// TIA Portal V20 program export: 1 tag tables, 0 data types, 2 data blocks, 4 code blocks (in call order from the OBs), 4 instance data blocks

VAR_GLOBAL   // PLC tag table "默认变量表"
   取芯V90_Actor_Interface_AddressIn AT %I82.0 : "PD_TEL3_IN";
   取芯V90_Actor_Interface_AddressOut AT %Q74.0 : "PD_TEL3_OUT";
   纠偏V90_Actor_Interface_AddressIn AT %I64.0 : "PD_TEL3_IN";
   纠偏V90_Actor_Interface_AddressOut AT %Q64.0 : "PD_TEL3_OUT";
   System_Byte AT %MB1 : Byte;
   FirstScan AT %M1.0 : Bool;
   DiagStatusUpdate AT %M1.1 : Bool;
   AlwaysTRUE AT %M1.2 : Bool;
   AlwaysFALSE AT %M1.3 : Bool;
   Clock_Byte AT %MB0 : Byte;
   Clock_10Hz AT %M0.0 : Bool;
   Clock_5Hz AT %M0.1 : Bool;
   "Clock_2.5Hz" AT %M0.2 : Bool;
   Clock_2Hz AT %M0.3 : Bool;
   "Clock_1.25Hz" AT %M0.4 : Bool;
   Clock_1Hz AT %M0.5 : Bool;
   "Clock_0.625Hz" AT %M0.6 : Bool;
   "Clock_0.5Hz" AT %M0.7 : Bool;
   纠偏V90控制字 AT %MW2 : Word;
   纠偏V90状态字 AT %MW4 : Word;
   纠_回原模式 AT %MW6 : Int;
   纠_绝对位置 AT %MD8 : Real;
   纠_相对位置 AT %MD12 : Real;
   纠_绝对速度 AT %MD16 : Real;
   纠_点动速度 AT %MD20 : Real;
   纠_当前位置 AT %M24.0 : LReal;
   纠_当前速度 AT %M32.0 : LReal;
   取芯V90控制字 AT %MW40 : Word;
   取芯V90状态字 AT %MW42 : Word;
   取_回原模式 AT %MW44 : Int;
   取_绝对位置 AT %MD46 : Real;
   取_绝对速度 AT %MD50 : Real;
   取_相对位置 AT %MD54 : Real;
   取_相对速度 AT %MD58 : Real;
   取_点动速度 AT %MD62 : Real;
   取_当前速度 AT %M66.0 : LReal;
   取_当前位置 AT %M74.0 : LReal;
END_VAR

DATA_BLOCK "G2_上传"   // DB2
{ S7_Optimized_Access := 'FALSE' }
   VAR
      位1 : Bool;
      位2 : Bool;
      位3 : Bool;
      位4 : Bool;
      位5 : Bool;
      位6 : Bool;
      位7 : Bool;
      位8 : Bool;
      位9 : Bool;
      位10 : Bool;
      位11 : Bool;
      位12 : Bool;
      位13 : Bool;
      位14 : Bool;
      位15 : Bool;
      位16 : Bool;
      位17 : Bool;
      位18 : Bool;
      位19 : Bool;
      位20 : Bool;
      位21 : Bool;
      位22 : Bool;
      位23 : Bool;
      位24 : Bool;
      位25 : Bool;
      位26 : Bool;
      位27 : Bool;
      位28 : Bool;
      位29 : Bool;
      位30 : Bool;
      整型1 : Int;
      整型2 : Int;
      整型3 : Int;
      整型4 : Int;
      整型5 : Int;
      整型6 : Int;
      整型7 : Int;
      整型8 : Int;
      整型9 : Int;
      整型10 : Int;
      浮点数1 : Real;
      浮点数2 : Real;
      浮点数3 : Real;
      浮点数4 : Real;
      浮点数5 : Real;
      浮点数6 : Real;
      浮点数7 : Real;
      浮点数8 : Real;
      浮点数9 : Real;
      浮点数10 : Real;
      浮点数11 : Real;
      浮点数12 : Real;
      浮点数13 : Real;
      浮点数14 : Real;
      浮点数15 : Real;
      浮点数16 : Real;
      浮点数17 : Real;
      浮点数18 : Real;
      浮点数19 : Real;
   END_VAR
BEGIN
END_DATA_BLOCK

DATA_BLOCK "G2_下载"   // DB1
{ S7_Optimized_Access := 'FALSE' }
   VAR
      位1 : Bool;
      位2 : Bool;
      位3 : Bool;
      位4 : Bool;
      位5 : Bool;
      位6 : Bool;
      位7 : Bool;
      位8 : Bool;
      位9 : Bool;
      位10 : Bool;
      位11 : Bool;
      位12 : Bool;
      位13 : Bool;
      位14 : Bool;
      位15 : Bool;
      位16 : Bool;
      位17 : Bool;
      位18 : Bool;
      位19 : Bool;
      位20 : Bool;
      位21 : Bool;
      位22 : Bool;
      位23 : Bool;
      位24 : Bool;
      位25 : Bool;
      位26 : Bool;
      位27 : Bool;
      位28 : Bool;
      位29 : Bool;
      位30 : Bool;
      整型1 : Int;
      整型2 : Int;
      整型3 : Int;
      整型4 : Int;
      整型5 : Int;
      整型6 : Int;
      整型7 : Int;
      整型8 : Int;
      整型9 : Int;
      整型10 : Int;
      浮点数1 : Real;
      浮点数2 : Real;
      浮点数3 : Real;
      浮点数4 : Real;
      浮点数5 : Real;
      浮点数6 : Real;
      浮点数7 : Real;
      浮点数8 : Real;
      浮点数9 : Real;
      浮点数10 : Real;
      浮点数11 : Real;
      浮点数12 : Real;
      浮点数13 : Real;
      浮点数14 : Real;
      浮点数15 : Real;
      浮点数16 : Real;
      浮点数17 : Real;
      浮点数18 : Real;
      浮点数19 : Real;
   END_VAR
BEGIN
END_DATA_BLOCK

ORGANIZATION_BLOCK "Main"   // OB1, LAD, ProgramCycle
TITLE = "Main Program Sweep (Cycle)"
{ S7_Optimized_Access := 'TRUE' }
// stored: SetENOAutomatically false
   VAR_INPUT
      Initial_Call : Bool;   // Initial call of this OB
      Remanence : Bool;   // =True, if remanent data are available
   END_VAR
BEGIN
END_ORGANIZATION_BLOCK

FUNCTION_BLOCK "定位轴基本控制"   // FB1, LAD
{ S7_Optimized_Access := 'TRUE' }
// stored: MemoryReserve 100, SetENOAutomatically false
   VAR_INPUT
      轴号 : TO_PositioningAxis;
      使能 : Bool;
      回原 : Bool;
      回原模式 : Int;
      绝对定位 : Bool;
      相对定位 : Bool;
      暂停 : Bool;
      复位 : Bool;
      绝对位置 : Real;
      绝对速度 : Real;
      相对位置 : Real;
      相对速度 : Real;
      点动正转 : Bool;
      点动反转 : Bool;
      点动速度 : Real;
   END_VAR
   VAR_OUTPUT
      轴已启用 : Bool;
      使能错误 : Bool;
      回原完成 : Bool;
      回原错误 : Bool;
      绝对定位完成 : Bool;
      绝对定位错误 : Bool;
      相对定位完成 : Bool;
      相对定位错误 : Bool;
      点动中 : Bool;
      点动错误 : Bool;
      当前位置 : LReal;
      当前速度 : LReal;
   END_VAR
   VAR
      MC_Power_Instance { S7_SetPoint := 'True'} : MC_POWER;
      MC_Home_Instance { S7_SetPoint := 'True'} : MC_HOME;
      MC_MoveAbsolute_Instance { S7_SetPoint := 'True'} : MC_MOVEABSOLUTE;
      MC_MoveRelative_Instance { S7_SetPoint := 'True'} : MC_MOVERELATIVE;
      MC_Reset_Instance { S7_SetPoint := 'True'} : MC_RESET;
      MC_Halt_Instance { S7_SetPoint := 'True'} : MC_HALT;
      MC_MoveJog_Instance { S7_SetPoint := 'True'} : MC_MOVEJOG;
   END_VAR
   VAR_TEMP
      复位完成 : Bool;
      复位错误 : Bool;
      暂停完成 : Bool;
      暂停错误 : Bool;
   END_VAR
   VAR_TEMP   // added for the SCL form of the ladder/FBD networks
      _w1 : Bool;
      _w2 : Bool;
      _w3 : Bool;
   END_VAR
BEGIN

REGION Network 1
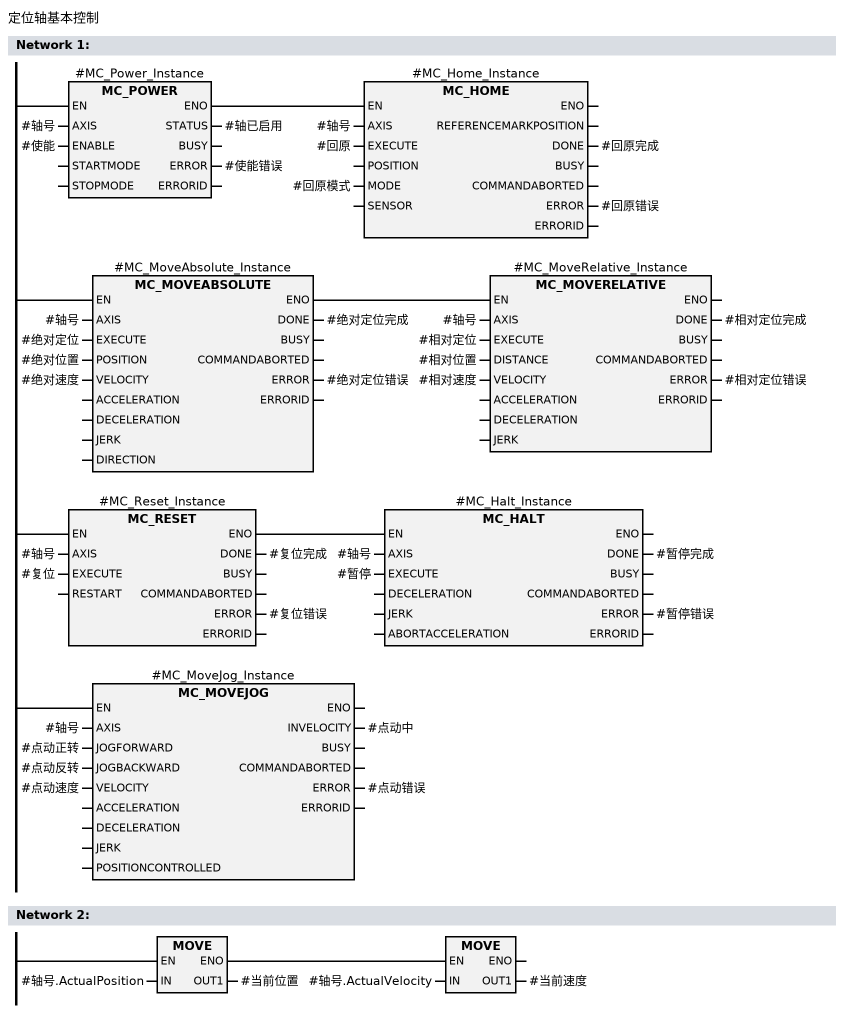
   RUNG wire#powerrail
      #MC_Power_Instance.MC_POWER(Axis := #轴号, Enable := #使能, StartMode :=, StopMode :=, Status => #轴已启用, Busy =>, Error => #使能错误, ErrorId =>)
      #MC_Home_Instance.MC_HOME(Axis := #轴号, Execute := #回原, Position :=, Mode := #回原模式, Sensor :=, ReferenceMarkPosition =>, Done => #回原完成, Busy =>, CommandAborted =>, Error => #回原错误, ErrorId =>)
   END_RUNG
   RUNG wire#powerrail
      #MC_MoveAbsolute_Instance.MC_MOVEABSOLUTE(Axis := #轴号, Execute := #绝对定位, Position := #绝对位置, Velocity := #绝对速度, Acceleration :=, Deceleration :=, Jerk :=, Direction :=, Done => #绝对定位完成, Busy =>, CommandAborted =>, Error => #绝对定位错误, ErrorId =>)
      #MC_MoveRelative_Instance.MC_MOVERELATIVE(Axis := #轴号, Execute := #相对定位, Distance := #相对位置, Velocity := #相对速度, Acceleration :=, Deceleration :=, Jerk :=, Done => #相对定位完成, Busy =>, CommandAborted =>, Error => #相对定位错误, ErrorId =>)
   END_RUNG
   RUNG wire#powerrail
      #MC_Reset_Instance.MC_RESET(Axis := #轴号, Execute := #复位, Restart :=, Done => #复位完成, Busy =>, CommandAborted =>, Error => #复位错误, ErrorId =>)
      #MC_Halt_Instance.MC_HALT(Axis := #轴号, Execute := #暂停, Deceleration :=, Jerk :=, AbortAcceleration :=, Done => #暂停完成, Busy =>, CommandAborted =>, Error => #暂停错误, ErrorId =>)
   END_RUNG
   RUNG wire#powerrail
      #MC_MoveJog_Instance.MC_MOVEJOG(Axis := #轴号, JogForward := #点动正转, JogBackward := #点动反转, Velocity := #点动速度, Acceleration :=, Deceleration :=, Jerk :=, PositionControlled :=, InVelocity => #点动中, Busy =>, CommandAborted =>, Error => #点动错误, ErrorId =>)
   END_RUNG
   // the same network as SCL:
   #MC_Power_Instance(Axis := #轴号, Enable := #使能, Status => #轴已启用, Error => #使能错误, ENO => #_w1);   // MC_POWER
   IF #_w1 THEN
       #MC_Home_Instance(Axis := #轴号, Execute := #回原, Mode := #回原模式, Done => #回原完成, Error => #回原错误);   // MC_HOME
   END_IF;
   #MC_MoveAbsolute_Instance(Axis := #轴号,   // MC_MOVEABSOLUTE
                           Execute := #绝对定位,
                           Position := #绝对位置,
                           Velocity := #绝对速度,
                           Done => #绝对定位完成,
                           Error => #绝对定位错误,
                           ENO => #_w2);
   IF #_w2 THEN
       #MC_MoveRelative_Instance(Axis := #轴号,   // MC_MOVERELATIVE
                               Execute := #相对定位,
                               Distance := #相对位置,
                               Velocity := #相对速度,
                               Done => #相对定位完成,
                               Error => #相对定位错误);
   END_IF;
   #MC_Reset_Instance(Axis := #轴号, Execute := #复位, Done => #复位完成, Error => #复位错误, ENO => #_w3);   // MC_RESET
   IF #_w3 THEN
       #MC_Halt_Instance(Axis := #轴号, Execute := #暂停, Done => #暂停完成, Error => #暂停错误);   // MC_HALT
   END_IF;
   #MC_MoveJog_Instance(Axis := #轴号,   // MC_MOVEJOG
                        JogForward := #点动正转,
                        JogBackward := #点动反转,
                        Velocity := #点动速度,
                        InVelocity => #点动中,
                        Error => #点动错误);
END_REGION

REGION Network 2
   RUNG wire#powerrail
      Move(in := #轴号.ActualPosition, out1 => #当前位置)
      Move(in := #轴号.ActualVelocity, out1 => #当前速度)
   END_RUNG
   // the same network as SCL:
   #当前位置 := #轴号.ActualPosition;
   #当前速度 := #轴号.ActualVelocity;
END_REGION
END_FUNCTION_BLOCK

FUNCTION "取芯伺服" : Void   // FC2, LAD
{ S7_Optimized_Access := 'TRUE' }
// stored: SetENOAutomatically false
BEGIN

REGION Network 1 (SCL)
   "取芯V90控制字".%X0 := "G2_下载".位9;
   "取芯V90控制字".%X1 := "G2_下载".位10;
   "取芯V90控制字".%X2 := "G2_下载".位11;
   "取芯V90控制字".%X3 := "G2_下载".位12;
   "取芯V90控制字".%X4 := "G2_下载".位13;
   "取芯V90控制字".%X5 := "G2_下载".位14;
   "取芯V90控制字".%X6 := "G2_下载".位15;
   "取芯V90控制字".%X7 := "G2_下载".位16;

   "取_回原模式" := "G2_下载".整型2;

   "取_绝对位置" := "G2_下载".浮点数6;
   "取_绝对速度" := "G2_下载".浮点数7;
   "取_相对位置" := "G2_下载".浮点数8;
   "取_相对位置" := "G2_下载".浮点数9;
   "取_点动速度" := "G2_下载".浮点数10;
END_REGION

REGION Network 2
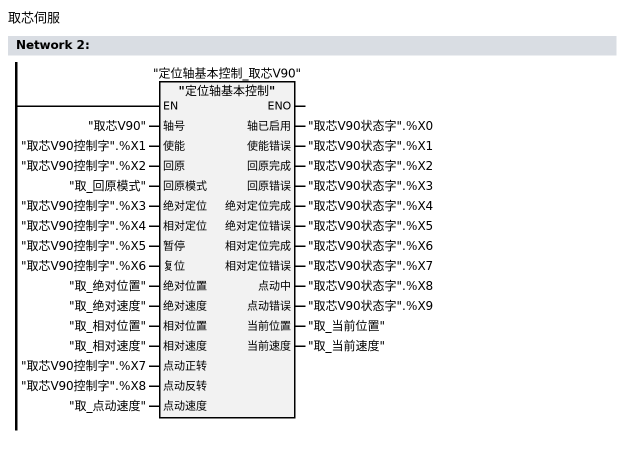
   RUNG wire#powerrail
      "定位轴基本控制_取芯V90"(轴号 := "取芯V90", 使能 := "取芯V90控制字".%X1, 回原 := "取芯V90控制字".%X2, 回原模式 := "取_回原模式", 绝对定位 := "取芯V90控制字".%X3, 相对定位 := "取芯V90控制字".%X4, 暂停 := "取芯V90控制字".%X5, 复位 := "取芯V90控制字".%X6, 绝对位置 := "取_绝对位置", 绝对速度 := "取_绝对速度", 相对位置 := "取_相对位置", 相对速度 := "取_相对速度", 点动正转 := "取芯V90控制字".%X7, 点动反转 := "取芯V90控制字".%X8, 点动速度 := "取_点动速度", 轴已启用 => "取芯V90状态字".%X0, 使能错误 => "取芯V90状态字".%X1, 回原完成 => "取芯V90状态字".%X2, 回原错误 => "取芯V90状态字".%X3, 绝对定位完成 => "取芯V90状态字".%X4, 绝对定位错误 => "取芯V90状态字".%X5, 相对定位完成 => "取芯V90状态字".%X6, 相对定位错误 => "取芯V90状态字".%X7, 点动中 => "取芯V90状态字".%X8, 点动错误 => "取芯V90状态字".%X9, 当前位置 => "取_当前位置", 当前速度 => "取_当前速度")
   END_RUNG
   // the same network as SCL:
   "定位轴基本控制_取芯V90"(轴号 := "取芯V90",   // "定位轴基本控制"
                   使能 := "取芯V90控制字".%X1,
                   回原 := "取芯V90控制字".%X2,
                   回原模式 := "取_回原模式",
                   绝对定位 := "取芯V90控制字".%X3,
                   相对定位 := "取芯V90控制字".%X4,
                   暂停 := "取芯V90控制字".%X5,
                   复位 := "取芯V90控制字".%X6,
                   绝对位置 := "取_绝对位置",
                   绝对速度 := "取_绝对速度",
                   相对位置 := "取_相对位置",
                   相对速度 := "取_相对速度",
                   点动正转 := "取芯V90控制字".%X7,
                   点动反转 := "取芯V90控制字".%X8,
                   点动速度 := "取_点动速度",
                   轴已启用 => "取芯V90状态字".%X0,
                   使能错误 => "取芯V90状态字".%X1,
                   回原完成 => "取芯V90状态字".%X2,
                   回原错误 => "取芯V90状态字".%X3,
                   绝对定位完成 => "取芯V90状态字".%X4,
                   绝对定位错误 => "取芯V90状态字".%X5,
                   相对定位完成 => "取芯V90状态字".%X6,
                   相对定位错误 => "取芯V90状态字".%X7,
                   点动中 => "取芯V90状态字".%X8,
                   点动错误 => "取芯V90状态字".%X9,
                   当前位置 => "取_当前位置",
                   当前速度 => "取_当前速度");
END_REGION

REGION Network 3 (SCL)
   "G2_上传".位11 := "取芯V90状态字".%X0;
   "G2_上传".位12 := "取芯V90状态字".%X1;
   "G2_上传".位13 := "取芯V90状态字".%X2;
   "G2_上传".位14 := "取芯V90状态字".%X3;
   "G2_上传".位15 := "取芯V90状态字".%X4;
   "G2_上传".位16 := "取芯V90状态字".%X5;
   "G2_上传".位17 := "取芯V90状态字".%X6;
   "G2_上传".位18 := "取芯V90状态字".%X7;
   "G2_上传".位19 := "取芯V90状态字".%X8;
   "G2_上传".位20 := "取芯V90状态字".%X9;

   "G2_上传".浮点数3 := LREAL_TO_REAL(IN := "取_当前位置");
   "G2_上传".浮点数4 := LREAL_TO_REAL(IN := "取_当前速度");
END_REGION
END_FUNCTION

FUNCTION "纠偏伺服" : Void   // FC1, LAD
{ S7_Optimized_Access := 'TRUE' }
// stored: SetENOAutomatically false
BEGIN

REGION Network 1 (SCL)
   "纠偏V90控制字".%X0:="G2_下载".位1;
   "纠偏V90控制字".%X1 := "G2_下载".位2;
   "纠偏V90控制字".%X2 := "G2_下载".位3;
   "纠偏V90控制字".%X3 := "G2_下载".位4;
   "纠偏V90控制字".%X4 := "G2_下载".位5;
   "纠偏V90控制字".%X5 := "G2_下载".位6;
   "纠偏V90控制字".%X6 := "G2_下载".位7;
   "纠偏V90控制字".%X7 := "G2_下载".位8;

   "纠_回原模式" := "G2_下载".整型1;

   "纠_绝对位置" := "G2_下载".浮点数1;
   "纠_绝对速度" := "G2_下载".浮点数2;
   "纠_相对位置" := "G2_下载".浮点数3;
   "纠_相对位置" := "G2_下载".浮点数4;
   "纠_点动速度" := "G2_下载".浮点数5;
END_REGION

REGION Network 2
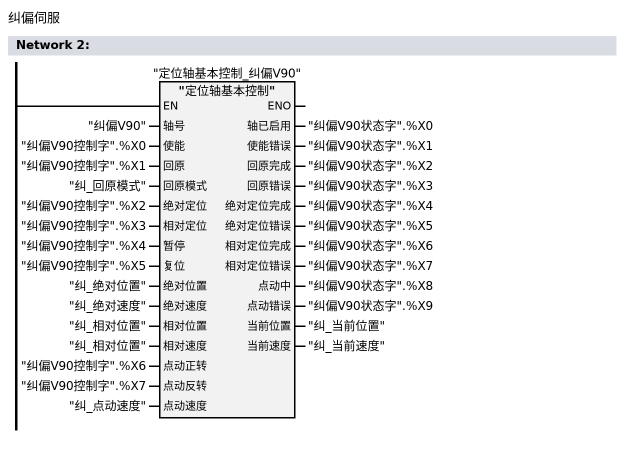
   RUNG wire#powerrail
      "定位轴基本控制_纠偏V90"(轴号 := "纠偏V90", 使能 := "纠偏V90控制字".%X0, 回原 := "纠偏V90控制字".%X1, 回原模式 := "纠_回原模式", 绝对定位 := "纠偏V90控制字".%X2, 相对定位 := "纠偏V90控制字".%X3, 暂停 := "纠偏V90控制字".%X4, 复位 := "纠偏V90控制字".%X5, 绝对位置 := "纠_绝对位置", 绝对速度 := "纠_绝对速度", 相对位置 := "纠_相对位置", 相对速度 := "纠_相对位置", 点动正转 := "纠偏V90控制字".%X6, 点动反转 := "纠偏V90控制字".%X7, 点动速度 := "纠_点动速度", 轴已启用 => "纠偏V90状态字".%X0, 使能错误 => "纠偏V90状态字".%X1, 回原完成 => "纠偏V90状态字".%X2, 回原错误 => "纠偏V90状态字".%X3, 绝对定位完成 => "纠偏V90状态字".%X4, 绝对定位错误 => "纠偏V90状态字".%X5, 相对定位完成 => "纠偏V90状态字".%X6, 相对定位错误 => "纠偏V90状态字".%X7, 点动中 => "纠偏V90状态字".%X8, 点动错误 => "纠偏V90状态字".%X9, 当前位置 => "纠_当前位置", 当前速度 => "纠_当前速度")
   END_RUNG
   // the same network as SCL:
   "定位轴基本控制_纠偏V90"(轴号 := "纠偏V90",   // "定位轴基本控制"
                   使能 := "纠偏V90控制字".%X0,
                   回原 := "纠偏V90控制字".%X1,
                   回原模式 := "纠_回原模式",
                   绝对定位 := "纠偏V90控制字".%X2,
                   相对定位 := "纠偏V90控制字".%X3,
                   暂停 := "纠偏V90控制字".%X4,
                   复位 := "纠偏V90控制字".%X5,
                   绝对位置 := "纠_绝对位置",
                   绝对速度 := "纠_绝对速度",
                   相对位置 := "纠_相对位置",
                   相对速度 := "纠_相对位置",
                   点动正转 := "纠偏V90控制字".%X6,
                   点动反转 := "纠偏V90控制字".%X7,
                   点动速度 := "纠_点动速度",
                   轴已启用 => "纠偏V90状态字".%X0,
                   使能错误 => "纠偏V90状态字".%X1,
                   回原完成 => "纠偏V90状态字".%X2,
                   回原错误 => "纠偏V90状态字".%X3,
                   绝对定位完成 => "纠偏V90状态字".%X4,
                   绝对定位错误 => "纠偏V90状态字".%X5,
                   相对定位完成 => "纠偏V90状态字".%X6,
                   相对定位错误 => "纠偏V90状态字".%X7,
                   点动中 => "纠偏V90状态字".%X8,
                   点动错误 => "纠偏V90状态字".%X9,
                   当前位置 => "纠_当前位置",
                   当前速度 => "纠_当前速度");
END_REGION

REGION Network 3 (SCL)
   "G2_上传".位1 := "纠偏V90状态字".%X0;
   "G2_上传".位2 := "纠偏V90状态字".%X1;
   "G2_上传".位3 := "纠偏V90状态字".%X2;
   "G2_上传".位4 := "纠偏V90状态字".%X3;
   "G2_上传".位5 := "纠偏V90状态字".%X4;
   "G2_上传".位6 := "纠偏V90状态字".%X5;
   "G2_上传".位7 := "纠偏V90状态字".%X6;
   "G2_上传".位8 := "纠偏V90状态字".%X7;
   "G2_上传".位9 := "纠偏V90状态字".%X8;
   "G2_上传".位10 := "纠偏V90状态字".%X9;

   "G2_上传".浮点数1 := LREAL_TO_REAL(IN := "纠_当前位置");
   "G2_上传".浮点数2 := LREAL_TO_REAL(IN := "纠_当前速度");
END_REGION
END_FUNCTION

DATA_BLOCK "定位轴基本控制_取芯V90"   // DB6
// stored: InstanceOfName 定位轴基本控制, InstanceOfType FB
"定位轴基本控制"
BEGIN
END_DATA_BLOCK

DATA_BLOCK "定位轴基本控制_纠偏V90"   // DB5
// stored: InstanceOfName 定位轴基本控制, InstanceOfType FB
"定位轴基本控制"
BEGIN
END_DATA_BLOCK

DATA_BLOCK "取芯V90"   // DB3, Motion_DB
// stored: InstanceOfName TO_PositioningAxis, OfSystemLibElement TO_PositioningAxis, OfSystemLibVersion 8.0
TO_PositioningAxis   // technology object, version 8.0
// stored: Connection Interface Actor, InputAddress 656, OutputAddress 592
// stored: Connection Interface Sensor[1], InputAddress 656, OutputAddress 592, SensorIndexInActorTelegram 1
   // // inherited from TO_SpeedAxis
   // // inherited from TO_Axis
   // // inherited from TO_Object
   // VAR
   //    Actor : TO_Struct_Actor;
   // END_VAR
   // VAR
   //    Position { ExternalWritable := 'False'} : LReal;
   //    ActualPosition { ExternalWritable := 'False'} : LReal;
   //    ActualVelocity { ExternalWritable := 'False'} : LReal;
   //    ActualAcceleration { ExternalWritable := 'False'} : LReal;
   //    OperativeSensor { ExternalWritable := 'False'} : UDInt;
   //    ModuloCycle { ExternalWritable := 'False'} : DInt;
   //    ActualModuloCycle { ExternalWritable := 'False'} : DInt;
   //    Sensor { S7_SetPoint := 'True'} : Array[1..4] of TO_Struct_Sensor;
   //    Extrapolation { S7_SetPoint := 'True'} : TO_Struct_Extrapolation;
   //    Mechanics { S7_SetPoint := 'True'} : TO_Struct_Mechanics;
   //    Properties { ExternalWritable := 'False'; S7_SetPoint := 'True'} : TO_Struct_Properties;
   //    Modulo { S7_SetPoint := 'True'} : TO_Struct_Modulo;
   //    PositionLimits_SW { S7_SetPoint := 'True'} : TO_Struct_PositionLimitsSW;
   //    PositionLimits_HW { S7_SetPoint := 'True'} : TO_Struct_PositionLimitsHW;
   //    Homing { S7_SetPoint := 'True'} : TO_Struct_Homing;
   //    PositionControl { S7_SetPoint := 'True'} : TO_Struct_PositionControl;
   //    SetpointFilter { S7_SetPoint := 'True'} : TO_Struct_SetpointFilter;
   //    DynamicAxisModel { S7_SetPoint := 'True'} : TO_Struct_DynamicAxisModel;
   //    FollowingError { S7_SetPoint := 'True'} : TO_Struct_FollowingError;
   //    PositioningMonitoring { S7_SetPoint := 'True'} : TO_Struct_PositioningMonitoring;
   //    StandstillSignal { S7_SetPoint := 'True'} : TO_Struct_StandstillSignal;
   //    StatusPositioning { ExternalWritable := 'False'; S7_SetPoint := 'True'} : TO_Struct_StatusPositioning;
   //    StatusServo { ExternalWritable := 'False'; S7_SetPoint := 'True'} : TO_Struct_StatusServo;
   //    StatusProvidedLeadingValue { ExternalWritable := 'False'; S7_SetPoint := 'True'} : TO_Struct_StatusProvidedLeadingValue;
   //    StatusSensor { ExternalWritable := 'False'; S7_SetPoint := 'True'} : Array[1..4] of TO_Struct_StatusSensor;
   //    StatusExtrapolation { ExternalWritable := 'False'; S7_SetPoint := 'True'} : TO_Struct_StatusExtrapolation;
   //    StatusKinematicsMotion { ExternalWritable := 'False'; S7_SetPoint := 'True'} : TO_Struct_StatusKinematicsMotion;
   // END_VAR
BEGIN
   Actor.Interface.AddressIn.RID := 16#208070c;
   Actor.Interface.AddressIn.AREA := 16#81;
   Actor.Interface.AddressIn.OFFSET := 656;
   Actor.Interface.AddressOut.RID := 16#208070d;
   Actor.Interface.AddressOut.AREA := 16#82;
   Actor.Interface.AddressOut.OFFSET := 592;
   Sensor[1].Interface.AddressIn.RID := 16#208070c;
   Sensor[1].Interface.AddressIn.AREA := 16#81;
   Sensor[1].Interface.AddressIn.OFFSET := 656;
   Sensor[1].Interface.AddressOut.RID := 16#208070d;
   Sensor[1].Interface.AddressOut.AREA := 16#82;
   Sensor[1].Interface.AddressOut.OFFSET := 592;
   _Actor.Interface.Telegram := 3;
   _Sensor[1].Interface.Telegram := 3;
END_DATA_BLOCK

DATA_BLOCK "纠偏V90"   // DB4, Motion_DB
// stored: InstanceOfName TO_PositioningAxis, OfSystemLibElement TO_PositioningAxis, OfSystemLibVersion 8.0
TO_PositioningAxis   // technology object, version 8.0
// stored: Connection Interface Actor, InputAddress 512, OutputAddress 512
// stored: Connection Interface Sensor[1], InputAddress 512, OutputAddress 512, SensorIndexInActorTelegram 1
   // // inherited from TO_SpeedAxis
   // // inherited from TO_Axis
   // // inherited from TO_Object
   // VAR
   //    Actor : TO_Struct_Actor;
   // END_VAR
   // VAR
   //    Position { ExternalWritable := 'False'} : LReal;
   //    ActualPosition { ExternalWritable := 'False'} : LReal;
   //    ActualVelocity { ExternalWritable := 'False'} : LReal;
   //    ActualAcceleration { ExternalWritable := 'False'} : LReal;
   //    OperativeSensor { ExternalWritable := 'False'} : UDInt;
   //    ModuloCycle { ExternalWritable := 'False'} : DInt;
   //    ActualModuloCycle { ExternalWritable := 'False'} : DInt;
   //    Sensor { S7_SetPoint := 'True'} : Array[1..4] of TO_Struct_Sensor;
   //    Extrapolation { S7_SetPoint := 'True'} : TO_Struct_Extrapolation;
   //    Mechanics { S7_SetPoint := 'True'} : TO_Struct_Mechanics;
   //    Properties { ExternalWritable := 'False'; S7_SetPoint := 'True'} : TO_Struct_Properties;
   //    Modulo { S7_SetPoint := 'True'} : TO_Struct_Modulo;
   //    PositionLimits_SW { S7_SetPoint := 'True'} : TO_Struct_PositionLimitsSW;
   //    PositionLimits_HW { S7_SetPoint := 'True'} : TO_Struct_PositionLimitsHW;
   //    Homing { S7_SetPoint := 'True'} : TO_Struct_Homing;
   //    PositionControl { S7_SetPoint := 'True'} : TO_Struct_PositionControl;
   //    SetpointFilter { S7_SetPoint := 'True'} : TO_Struct_SetpointFilter;
   //    DynamicAxisModel { S7_SetPoint := 'True'} : TO_Struct_DynamicAxisModel;
   //    FollowingError { S7_SetPoint := 'True'} : TO_Struct_FollowingError;
   //    PositioningMonitoring { S7_SetPoint := 'True'} : TO_Struct_PositioningMonitoring;
   //    StandstillSignal { S7_SetPoint := 'True'} : TO_Struct_StandstillSignal;
   //    StatusPositioning { ExternalWritable := 'False'; S7_SetPoint := 'True'} : TO_Struct_StatusPositioning;
   //    StatusServo { ExternalWritable := 'False'; S7_SetPoint := 'True'} : TO_Struct_StatusServo;
   //    StatusProvidedLeadingValue { ExternalWritable := 'False'; S7_SetPoint := 'True'} : TO_Struct_StatusProvidedLeadingValue;
   //    StatusSensor { ExternalWritable := 'False'; S7_SetPoint := 'True'} : Array[1..4] of TO_Struct_StatusSensor;
   //    StatusExtrapolation { ExternalWritable := 'False'; S7_SetPoint := 'True'} : TO_Struct_StatusExtrapolation;
   //    StatusKinematicsMotion { ExternalWritable := 'False'; S7_SetPoint := 'True'} : TO_Struct_StatusKinematicsMotion;
   // END_VAR
BEGIN
   Actor.Interface.AddressIn.RID := 16#208070c;
   Actor.Interface.AddressIn.AREA := 16#81;
   Actor.Interface.AddressIn.OFFSET := 512;
   Actor.Interface.AddressOut.RID := 16#208070d;
   Actor.Interface.AddressOut.AREA := 16#82;
   Actor.Interface.AddressOut.OFFSET := 512;
   Sensor[1].Interface.AddressIn.RID := 16#208070c;
   Sensor[1].Interface.AddressIn.AREA := 16#81;
   Sensor[1].Interface.AddressIn.OFFSET := 512;
   Sensor[1].Interface.AddressOut.RID := 16#208070d;
   Sensor[1].Interface.AddressOut.AREA := 16#82;
   Sensor[1].Interface.AddressOut.OFFSET := 512;
   _Actor.Interface.Telegram := 3;
   _Sensor[1].Interface.Telegram := 3;
END_DATA_BLOCK
